FUNCTION_BLOCK PUBLIC FB_LampSetLevelCommand IMPLEMENTS I_Command
VAR
	refLamp		: REFERENCE TO FB_Lamp;
	byNewLevel	: BYTE;
	byLastLevel : BYTE := 255;
END_VAR

METHOD Execute
IF (__ISVALIDREF(THIS^.refLamp)) THEN
	THIS^.byLastLevel := THIS^.refLamp.Level;	
	THIS^.refLamp.SetLevel(THIS^.byNewLevel);
END_IF
END_METHOD

METHOD FB_init : BOOL
VAR_INPUT
	bInitRetains : BOOL; // if TRUE, the retain variables are initialized (warm start / cold start)
	bInCopyCode : BOOL;  // if TRUE, the instance afterwards gets moved into the copy code (online change)
	refLamp : REFERENCE TO FB_Lamp;
	byNewLevel : BYTE;
END_VAR
IF (__ISVALIDREF(refLamp)) THEN
	THIS^.refLamp REF= refLamp;
ELSE
	THIS^.refLamp REF= 0;
END_IF
THIS^.byNewLevel := byNewLevel;
END_METHOD

METHOD Undo
IF (__ISVALIDREF(THIS^.refLamp)) THEN
	IF (THIS^.byLastLevel <> 255) THEN
		THIS^.refLamp.SetLevel(THIS^.byLastLevel);
	END_IF
END_IF
END_METHOD

END_FUNCTION_BLOCK

(* stored: Version 1.1.0.1, ProductVersion 3.1.4020.3
   POU FB_LampSetLevelCommand: Id {9f6e262f-5575-454c-8f85-b9e06af108eb}, SpecialFunc None
   Method Execute: Id {d3314861-d094-46fb-bd7f-18bce7e27134}
   Method FB_init: Id {70db96a3-729e-4e7f-bbee-0bb72b3ab88e}
   Method Undo: Id {7c9a30e9-c779-4432-a51a-0fb35f3ba6e0} *)
